PROGRAM MAIN
VAR
	{ attribute 'TcHmiSymbol.AddSymbol' }
	nCtx			: DINT;
	
	{ attribute 'My.Custom.Attribute' }
	{ attribute 'TcHmiSymbol.AddSymbol' }
	nAttribute		: DINT;
	
END_VAR

END_PROGRAM

(* stored: Version 1.1.0.1
   POU MAIN: Id {28507b62-cd61-4eba-97c0-4dd3a4048b0c}, SpecialFunc None *)
